FUNCTION_BLOCK FB_Conveyor
VAR_INPUT
	
END_VAR
VAR_OUTPUT
END_VAR
VAR
	on : BOOL;
	timer0_emitter : Tc2_Standard.TP;
	EmitterTrigger : BOOL;
	Timer1 : Tc2_Standard.TON;
	Step_0_Standby : BOOL;
	Step_1 : BOOL;
	Step_2 : BOOL;
	Step_3 : BOOL;
	Step_4 : BOOL;
	Step_5 : BOOL;
	Step_6 : BOOL;
	Step_7 : BOOL;
	Step_10 : BOOL;
	Step_15 : BOOL;
	step_last : BOOL;
	
	condition : BOOL;
	
	Opstart_puls_OS : BOOL;

	
	Initialiser_SQ: BOOL;
END_VAR
VAR_IN_OUT
	control_data : PlantAndCMs.Udt_PlantControl_Mode_1;
	
	control_data_vision : CM_Vision_UDT;
	control_data_Conveyor1 : CM_DO_UDT;
	
	control_data_StopBlade : CM_DO_UDT;
	control_data_emitter : CM_DO_UDT;
END_VAR
VAR // added by the converter: edge detectors and wires of the graphical bodies
    _w1, _w2, _w3, _w4, _w5, _w6, _w7, _w8, _w9, _w10, _w11, _w12, _w13, _w14, _w15, _w16, _w17 : BOOL;
END_VAR

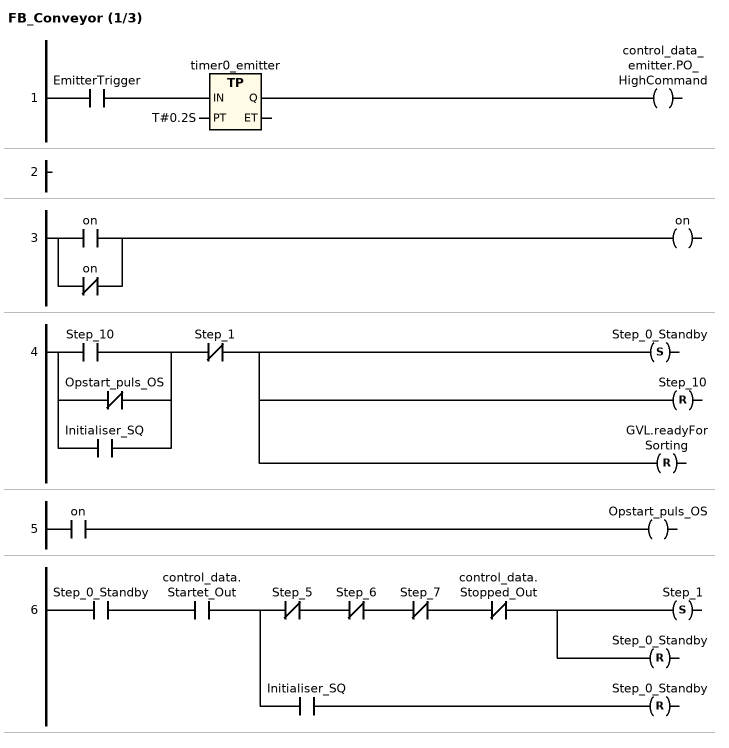
// NETWORK 1
timer0_emitter(IN := EmitterTrigger, PT := T#0.2S); // TP
control_data_emitter.PO_HighCommand := timer0_emitter.Q;

// NETWORK 2

// NETWORK 3
on := on OR NOT on;

// NETWORK 4
_w1 := (Step_10 OR NOT Opstart_puls_OS OR Initialiser_SQ) AND NOT Step_1;
Step_0_Standby S= _w1;
Step_10 R= _w1;
GVL.readyForSorting R= _w1;

// NETWORK 5
Opstart_puls_OS := on;

// NETWORK 6
_w2 := Step_0_Standby AND control_data.Startet_Out;
_w3 := _w2 AND NOT Step_5 AND NOT Step_6 AND NOT Step_7 AND NOT control_data.Stopped_Out;
Step_1 S= _w3;
Step_0_Standby R= _w3;
Step_0_Standby R= _w2 AND Initialiser_SQ;

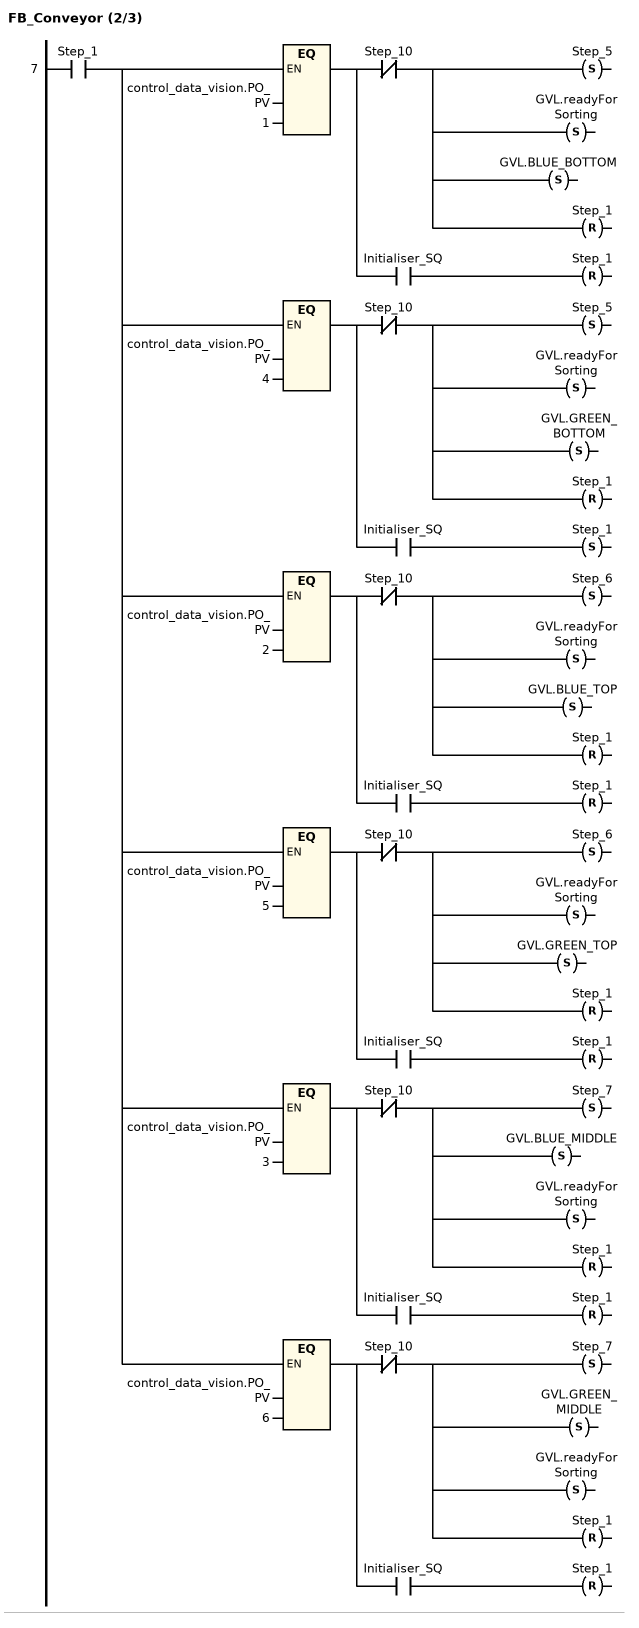
// NETWORK 7
_w4 := Step_1;
_w5 := _w4 AND control_data_vision.PO_PV = 1;
_w6 := _w5 AND NOT Step_10;
Step_5 S= _w6;
GVL.readyForSorting S= _w6;
GVL.BLUE_BOTTOM S= _w6;
Step_1 R= _w6;
Step_1 R= _w5 AND Initialiser_SQ;
_w7 := _w4 AND control_data_vision.PO_PV = 4;
_w8 := _w7 AND NOT Step_10;
Step_5 S= _w8;
GVL.readyForSorting S= _w8;
GVL.GREEN_BOTTOM S= _w8;
Step_1 R= _w8;
Step_1 S= _w7 AND Initialiser_SQ;
_w9 := _w4 AND control_data_vision.PO_PV = 2;
_w10 := _w9 AND NOT Step_10;
Step_6 S= _w10;
GVL.readyForSorting S= _w10;
GVL.BLUE_TOP S= _w10;
Step_1 R= _w10;
Step_1 R= _w9 AND Initialiser_SQ;
_w11 := _w4 AND control_data_vision.PO_PV = 5;
_w12 := _w11 AND NOT Step_10;
Step_6 S= _w12;
GVL.readyForSorting S= _w12;
GVL.GREEN_TOP S= _w12;
Step_1 R= _w12;
Step_1 R= _w11 AND Initialiser_SQ;
_w13 := _w4 AND control_data_vision.PO_PV = 3;
_w14 := _w13 AND NOT Step_10;
Step_7 S= _w14;
GVL.BLUE_MIDDLE S= _w14;
GVL.readyForSorting S= _w14;
Step_1 R= _w14;
Step_1 R= _w13 AND Initialiser_SQ;
_w15 := _w4 AND control_data_vision.PO_PV = 6;
_w16 := _w15 AND NOT Step_10;
Step_7 S= _w16;
GVL.GREEN_MIDDLE S= _w16;
GVL.readyForSorting S= _w16;
Step_1 R= _w16;
Step_1 R= _w15 AND Initialiser_SQ;

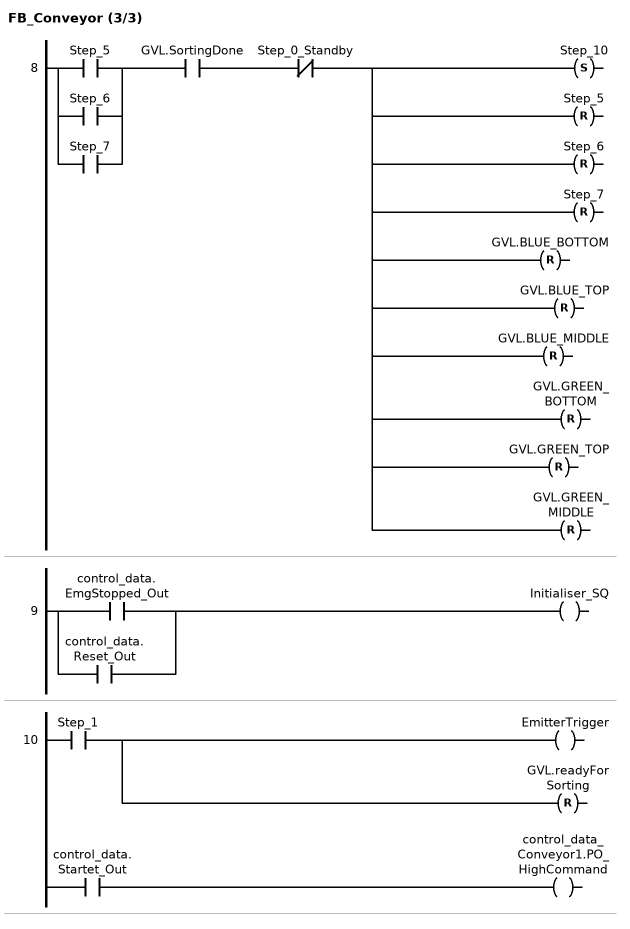
// NETWORK 8
_w17 := (Step_5 OR Step_6 OR Step_7) AND GVL.SortingDone AND NOT Step_0_Standby;
Step_10 S= _w17;
Step_5 R= _w17;
Step_6 R= _w17;
Step_7 R= _w17;
GVL.BLUE_BOTTOM R= _w17;
GVL.BLUE_TOP R= _w17;
GVL.BLUE_MIDDLE R= _w17;
GVL.GREEN_BOTTOM R= _w17;
GVL.GREEN_TOP R= _w17;
GVL.GREEN_MIDDLE R= _w17;

// NETWORK 9
Initialiser_SQ := control_data.EmgStopped_Out OR control_data.Reset_Out;

// NETWORK 10
EmitterTrigger := Step_1;
GVL.readyForSorting R= Step_1;
control_data_Conveyor1.PO_HighCommand := control_data.Startet_Out;

END_FUNCTION_BLOCK

(* stored: Version 1.1.0.1, ProductVersion 3.1.4024.13
   POU FB_Conveyor: Id {0cbf57b1-20ed-4dcc-924e-31c53c86553a}, SpecialFunc None *)
